SUBAPPLICATION front_fertilizer_main (* Subapplication Type *)
  (* Standard: 61499-2 *)
  (* Version 1.0, 2026-01-24, 04jul *)
  PACKAGE Main;
  IMPORT DefaultPool::Button_M1_refresh;
  IMPORT DefaultPool::Button_M1_reset;
  IMPORT DefaultPool::Button_M2_calibration_area_10a;
  IMPORT DefaultPool::Button_M2_calibration_area_1a;
  IMPORT DefaultPool::Button_M2_calibration_area_5a;
  IMPORT DefaultPool::Button_M2_start;
  IMPORT DefaultPool::Button_M4_manuel_start;
  IMPORT DefaultPool::Button_M4_manuel_stop;
  IMPORT DefaultPool::Button_W1_stop;
  IMPORT DefaultPool::Container_Picture_fertilzier_bin_empty_M1_filllevel;
  IMPORT DefaultPool::Container_Picture_fertilzier_bin_full_M1_filllevel;
  IMPORT DefaultPool::DataMask_M1;
  IMPORT DefaultPool::DataMask_M2;
  IMPORT DefaultPool::DataMask_M3;
  IMPORT DefaultPool::DataMask_M4;
  IMPORT DefaultPool::DataMask_M5;
  IMPORT DefaultPool::NumberVariable_D;
  IMPORT DefaultPool::NumberVariable_I;
  IMPORT DefaultPool::NumberVariable_P;
  IMPORT DefaultPool::NumberVariable_application_rate_percent;
  IMPORT DefaultPool::NumberVariable_engine_speed_manuel;
  IMPORT DefaultPool::NumberVariable_engine_speed_rpm;
  IMPORT DefaultPool::NumberVariable_flow_factor;
  IMPORT DefaultPool::NumberVariable_manuel_auto_speed;
  IMPORT DefaultPool::NumberVariable_selected_speed;
  IMPORT DefaultPool::NumberVariable_target_quantity;
  IMPORT DefaultPool::NumberVariable_target_quantity_calibration_run;
  IMPORT DefaultPool::OutputNumber_M1_weight;
  IMPORT DefaultPool::OutputString_M1_filllevel;
  IMPORT DefaultPool::SoftKeyMask_S1;
  IMPORT DefaultPool::SoftKeyMask_S2;
  IMPORT DefaultPool::SoftKeyMask_S3;
  IMPORT DefaultPool::SoftKeyMask_S4;
  IMPORT DefaultPool::SoftKey_100_percent;
  IMPORT DefaultPool::SoftKey_calibration_run;
  IMPORT DefaultPool::SoftKey_debug;
  IMPORT DefaultPool::SoftKey_main;
  IMPORT DefaultPool::SoftKey_minus_percent;
  IMPORT DefaultPool::SoftKey_plus_percent;
  IMPORT DefaultPool::SoftKey_settings;
  IMPORT DefaultPool::SoftKey_start;
  IMPORT DefaultPool::SoftKey_stop;
  IMPORT DefaultPool::WorkingSet_0;
  IMPORT Uebungen::const::NVS::NVS_Keys::KEY_I1_STORE;
  IMPORT Uebungen::const::NVS::NVS_Keys::KEY_I2_STORE;
  IMPORT Uebungen::const::NVS::NVS_Keys::KEY_I3_STORE;
  IMPORT Uebungen::const::NVS::NVS_Keys::SECTION_I1_STORE;
  IMPORT Uebungen::const::NVS::NVS_Keys::SECTION_I2_STORE;
  IMPORT Uebungen::const::NVS::NVS_Keys::SECTION_I3_STORE;
  IMPORT isobus::UT::Q::const::colours::COLOR_BLUE;
  IMPORT isobus::UT::Q::const::colours::COLOR_GREY;
  IMPORT isobus::UT::Q::const::colours::COLOR_RED;
  IMPORT isobus::UT::io::Button::ButtonActivationCode::BT_RELEASED_UNLATCHED;
  IMPORT isobus::UT::io::Softkey::SoftKeyActivationCode::SK_RELEASED;
  IMPORT logiBUS::io::AI::logiBUS_AI::AnalogInput_I6;
  IMPORT logiBUS::io::DI::logiBUS_DI::Input_I1;
  IMPORT logiBUS::io::DQ::logiBUS_DO::Output_Q2;
  IMPORT logiBUS::io::DQ::logiBUS_DO::Output_Q4;
  FBS
    Q_SoftKeyMask : isobus::UT::Q::Q_SoftKeyMask(u8MaskType := 1, u16DataMaskId := DataMask_M1, u16SoftKeyMaskId := SoftKeyMask_S1);
    Softkey_IE_main : isobus::UT::io::Softkey::Softkey_IE(QI := TRUE, u16ObjId := SoftKey_main, InputEvent := SK_RELEASED);
    Softkey_IE_calibration_run : isobus::UT::io::Softkey::Softkey_IE(QI := TRUE, u16ObjId := SoftKey_calibration_run, InputEvent := SK_RELEASED);
    Softkey_IE_settings : isobus::UT::io::Softkey::Softkey_IE(QI := TRUE, u16ObjId := SoftKey_settings, InputEvent := SK_RELEASED);
    Softkey_IE_debug : isobus::UT::io::Softkey::Softkey_IE(QI := TRUE, u16ObjId := SoftKey_debug, InputEvent := SK_RELEASED);
    Q_ActiveMask_DataMask_M1 : isobus::UT::Q::Q_ActiveMask(u16WorkSetId := WorkingSet_0);
    Q_NumericValue : isobus::UT::Q::Q_NumericValue(u16ObjId := NumberVariable_application_rate_percent);
    Softkey_IE_100_percent : isobus::UT::io::Softkey::Softkey_IE(QI := TRUE, u16ObjId := SoftKey_100_percent, InputEvent := SK_RELEASED);
    Softkey_IE_plus_percent : isobus::UT::io::Softkey::Softkey_IE(QI := TRUE, u16ObjId := SoftKey_plus_percent, InputEvent := SK_RELEASED);
    Softkey_IE_minus_percent : isobus::UT::io::Softkey::Softkey_IE(QI := TRUE, u16ObjId := SoftKey_minus_percent, InputEvent := SK_RELEASED);
    F_ADD : iec61131::arithmetic::F_ADD(IN2 := UDINT#278 (* Second function input *));
    F_SUB : iec61131::arithmetic::F_SUB(IN2 := UDINT#278 (* Second function input *));
    F_SEL_E_4 : eclipse4diac::utils::selection::F_SEL_E_4(IN1 := DataMask_M1, IN2 := DataMask_M2, IN3 := DataMask_M3, IN4 := DataMask_M4 (* Selectable input variable *));
    Q_ActiveMask_DataMask_M2 : isobus::UT::Q::Q_ActiveMask(u16WorkSetId := WorkingSet_0, u16NewMaskId := DataMask_M1);
    Q_SoftKeyMask_2 : isobus::UT::Q::Q_SoftKeyMask(u8MaskType := 1, u16DataMaskId := DataMask_M2, u16SoftKeyMaskId := SoftKeyMask_S2);
    Q_SoftKeyMask_3 : isobus::UT::Q::Q_SoftKeyMask(u8MaskType := 1, u16DataMaskId := DataMask_M3, u16SoftKeyMaskId := SoftKeyMask_S3);
    Q_SoftKeyMask_4 : isobus::UT::Q::Q_SoftKeyMask(u8MaskType := 1, u16DataMaskId := DataMask_M4, u16SoftKeyMaskId := SoftKeyMask_S4);
    F_SEL_E_3 : eclipse4diac::utils::selection::F_SEL_E_3(IN1 := UDINT#27780);
    NVS : eclipse4diac::storage::INI(QI := TRUE, SECTION := SECTION_I1_STORE, KEY := KEY_I1_STORE, DEFAULT_VALUE := UDINT#0);
    Q_NumericValue_1 : isobus::UT::Q::Q_NumericValue(u16ObjId := NumberVariable_application_rate_percent);
    CbVtStatus : isobus::UT::status::CbVtStatus;
    F_SEL_E_2 : eclipse4diac::utils::selection::F_SEL_E_2;
    Button_IE : isobus::UT::io::Button::Button_IE(QI := TRUE, u16ObjId := Button_M4_manuel_stop, InputEvent := BT_RELEASED_UNLATCHED);
    F_DWORD_TO_UDINT : iec61131::conversion::F_DWORD_TO_UDINT;
    InputNumber_I1 : isobus::UT::io::NumericValue::NumericValue_ID(QI := TRUE, u16ObjId := NumberVariable_flow_factor);
    INI : eclipse4diac::storage::INI(QI := TRUE, SECTION := SECTION_I2_STORE, KEY := KEY_I2_STORE, DEFAULT_VALUE := UDINT#55);
    Q_NumericValue_2 : isobus::UT::Q::Q_NumericValue(u16ObjId := NumberVariable_flow_factor);
    CbVtStatus_1 : isobus::UT::status::CbVtStatus;
    INI_1 : eclipse4diac::storage::INI(QI := TRUE, SECTION := SECTION_I3_STORE, KEY := KEY_I3_STORE, DEFAULT_VALUE := UDINT#55);
    CbVtStatus_2 : isobus::UT::status::CbVtStatus;
    F_DWORD_TO_UDINT_1 : iec61131::conversion::F_DWORD_TO_UDINT;
    InputNumber_I2 : isobus::UT::io::NumericValue::NumericValue_ID(QI := TRUE, u16ObjId := NumberVariable_target_quantity);
    Q_NumericValue_3 : isobus::UT::Q::Q_NumericValue(u16ObjId := NumberVariable_target_quantity);
    F_DINT_TO_UDINT : iec61131::conversion::F_DINT_TO_UDINT;
    F_DINT_TO_UDINT_1 : iec61131::conversion::F_DINT_TO_UDINT;
    F_DINT_TO_UDINT_2 : iec61131::conversion::F_DINT_TO_UDINT;
    logiBUS_IX : logiBUS::io::DI::logiBUS_IX(QI := True, Input := Input_I1);
    Q_StringValue : isobus::UT::Q::Q_StringValue(u16ObjId := OutputString_M1_filllevel);
    F_SEL : iec61131::selection::F_SEL(IN0 := STRING#'Tank leer', IN1 := STRING#'Tank voll');
    Q_ObjHideShow : isobus::UT::Q::Q_ObjHideShow(u16ObjId := Container_Picture_fertilzier_bin_full_M1_filllevel);
    Q_ObjHideShow_1 : isobus::UT::Q::Q_ObjHideShow(u16ObjId := Container_Picture_fertilzier_bin_empty_M1_filllevel);
    Q_BackgroundColour_3 : isobus::UT::Q::Q_BackgroundColour(u16ObjId := Button_M2_calibration_area_1a);
    Q_BackgroundColour_4 : isobus::UT::Q::Q_BackgroundColour(u16ObjId := Button_M2_calibration_area_5a);
    Q_BackgroundColour_5 : isobus::UT::Q::Q_BackgroundColour(u16ObjId := Button_M2_calibration_area_10a);
    F_SEL_E_5 : eclipse4diac::utils::selection::F_SEL_E_3(IN1 := COLOR_BLUE, IN2 := COLOR_GREY, IN3 := COLOR_GREY);
    F_SEL_E_6 : eclipse4diac::utils::selection::F_SEL_E_3(IN1 := COLOR_GREY, IN2 := COLOR_BLUE, IN3 := COLOR_GREY);
    Button_IE_1 : isobus::UT::io::Button::Button_IE(QI := TRUE, u16ObjId := Button_M2_calibration_area_1a, InputEvent := BT_RELEASED_UNLATCHED);
    Button_IE_2 : isobus::UT::io::Button::Button_IE(QI := TRUE, u16ObjId := Button_M2_calibration_area_5a, InputEvent := BT_RELEASED_UNLATCHED);
    Button_IE_3 : isobus::UT::io::Button::Button_IE(QI := TRUE, u16ObjId := Button_M2_calibration_area_10a, InputEvent := BT_RELEASED_UNLATCHED);
    F_SEL_E_7 : eclipse4diac::utils::selection::F_SEL_E_3(IN1 := COLOR_GREY, IN2 := COLOR_GREY, IN3 := COLOR_BLUE);
    Button_IE_4 : isobus::UT::io::Button::Button_IE(QI := TRUE, u16ObjId := Button_M2_start, InputEvent := BT_RELEASED_UNLATCHED);
    Q_ActiveMask_DataMask_M3 : isobus::UT::Q::Q_ActiveMask(u16WorkSetId := WorkingSet_0);
    F_SEL_E_8 : eclipse4diac::utils::selection::F_SEL_E_2(IN1 := DataMask_M5, IN2 := DataMask_M2);
    Button_IE_5 : isobus::UT::io::Button::Button_IE(QI := TRUE, u16ObjId := Button_W1_stop, InputEvent := BT_RELEASED_UNLATCHED);
    F_SEL_E_9 : eclipse4diac::utils::selection::F_SEL_E_3(IN1 := UDINT#100, IN2 := UDINT#20, IN3 := UDINT#10);
    F_DIV : iec61131::arithmetic::F_DIV;
    F_UDINT_TO_UINT : iec61131::conversion::F_UDINT_TO_UINT;
    Q_NumericValue_4 : isobus::UT::Q::Q_NumericValue(u16ObjId := NumberVariable_target_quantity_calibration_run);
    E_PERMIT : iec61499::events::E_PERMIT;
    E_SR : iec61499::events::E_SR;
    F_UDINT_TO_UINT_1 : iec61131::conversion::F_UDINT_TO_UINT;
    InputNumber_I3 : isobus::UT::io::NumericValue::NumericValue_ID(QI := TRUE, u16ObjId := NumberVariable_target_quantity);
    F_DWORD_TO_UDINT_2 : iec61131::conversion::F_DWORD_TO_UDINT;
    INI_2 : eclipse4diac::storage::INI(QI := TRUE, SECTION := SECTION_I3_STORE, KEY := KEY_I3_STORE, DEFAULT_VALUE := UDINT#55);
    Q_NumericValue_5 : isobus::UT::Q::Q_NumericValue(u16ObjId := NumberVariable_target_quantity);
    Softkey_IE_start : isobus::UT::io::Softkey::Softkey_IE(QI := TRUE, u16ObjId := SoftKey_start, InputEvent := SK_RELEASED);
    Softkey_IE_stop : isobus::UT::io::Softkey::Softkey_IE(QI := TRUE, u16ObjId := SoftKey_stop, InputEvent := SK_RELEASED);
    Q_BackgroundColour : isobus::UT::Q::Q_BackgroundColour(u16ObjId := SoftKey_start);
    Q_BackgroundColour_1 : isobus::UT::Q::Q_BackgroundColour(u16ObjId := SoftKey_stop);
    E_SR_1 : iec61499::events::E_SR;
    F_SEL_1 : iec61131::selection::F_SEL(IN0 := COLOR_BLUE, IN1 := COLOR_GREY);
    F_SEL_2 : iec61131::selection::F_SEL(IN0 := COLOR_GREY, IN1 := COLOR_RED);
    PWMOutput_Q4 : logiBUS::io::DQ::logiBUS_QD_PWM(QI := TRUE, OUT := 16#FFFFFFFF, Output := Output_Q4);
    AnalogInput_I6 : logiBUS::io::AI::logiBUS_AI_ID(QI := TRUE, Input := AnalogInput_I6, AnalogInput_hysteresis := 40);
    F_DWORD_TO_UDINT_3 : iec61131::conversion::F_DWORD_TO_UDINT;
    F_DWORD_TO_UDINT_4 : iec61131::conversion::F_DWORD_TO_UDINT;
    F_MUL : iec61131::arithmetic::F_MUL(IN2 := REAL#81.92);
    F_REAL_TO_UDINT : iec61131::conversion::F_REAL_TO_UDINT;
    F_UDINT_TO_REAL : iec61131::conversion::F_UDINT_TO_REAL;
    F_UDINT_TO_DWORD : iec61131::conversion::F_UDINT_TO_DWORD;
    F_LIMIT : iec61131::selection::F_LIMIT(MN := UDINT#0, MX := UDINT#8192);
    F_NOT : iec61131::bitwiseOperators::F_NOT;
    Button_IX : isobus::UT::io::Button::Button_IX(QI := TRUE, u16ObjId := Button_M1_reset);
    logiBUS_QX : logiBUS::io::DQ::logiBUS_QX(QI := TRUE, Output := Output_Q2);
    Q_NumericValue_6 : isobus::UT::Q::Q_NumericValue(u16ObjId := OutputNumber_M1_weight);
    E_DELAY : iec61499::events::E_DELAY(DT := T#2s);
    Button_IE_6 : isobus::UT::io::Button::Button_IE(QI := TRUE, u16ObjId := Button_M4_manuel_start, InputEvent := BT_RELEASED_UNLATCHED);
    NumericValue_ID : isobus::UT::io::NumericValue::NumericValue_ID(QI := TRUE, u16ObjId := NumberVariable_engine_speed_manuel);
    F_DWORD_TO_UDINT_5 : iec61131::conversion::F_DWORD_TO_UDINT;
    F_UDINT_TO_REAL_1 : iec61131::conversion::F_UDINT_TO_REAL;
    Q_NumericValue_7 : isobus::UT::Q::Q_NumericValue(u16ObjId := NumberVariable_engine_speed_rpm);
    F_REAL_TO_UDINT_1 : iec61131::conversion::F_REAL_TO_UDINT;
    Button_IE_7 : isobus::UT::io::Button::Button_IE(QI := TRUE, u16ObjId := Button_M1_refresh, InputEvent := BT_RELEASED_UNLATCHED);
    I_WBSD : isobus::tecu::I_WBSD(QI := TRUE);
    I_RHS : isobus::tecu::I_RHS(QI := TRUE);
    Q_NumericValue_8 : isobus::UT::Q::Q_NumericValue(u16ObjId := NumberVariable_selected_speed);
    F_UINT_TO_UDINT : iec61131::conversion::F_UINT_TO_UDINT;
    F_STRING_AS_BOOL : iec61131::conversion::F_STRING_AS_BOOL;
    F_BYTE_AS_STRING : iec61131::conversion::F_BYTE_AS_STRING;
    E_CYCLE : iec61499::events::E_CYCLE(DT := T#1s);
    NumericValue_ID_1 : isobus::UT::io::NumericValue::NumericValue_ID(QI := TRUE, u16ObjId := NumberVariable_P);
    F_DWORD_TO_UDINT_6 : iec61131::conversion::F_DWORD_TO_UDINT;
    F_UDINT_TO_REAL_2 : iec61131::conversion::F_UDINT_TO_REAL;
    NumericValue_ID_2 : isobus::UT::io::NumericValue::NumericValue_ID(QI := TRUE, u16ObjId := NumberVariable_I);
    F_DWORD_TO_UDINT_7 : iec61131::conversion::F_DWORD_TO_UDINT;
    F_UDINT_TO_REAL_3 : iec61131::conversion::F_UDINT_TO_REAL;
    NumericValue_ID_3 : isobus::UT::io::NumericValue::NumericValue_ID(QI := TRUE, u16ObjId := NumberVariable_D);
    F_DWORD_TO_UDINT_8 : iec61131::conversion::F_DWORD_TO_UDINT;
    F_UDINT_TO_REAL_4 : iec61131::conversion::F_UDINT_TO_REAL;
    NumericValue_ID_4 : isobus::UT::io::NumericValue::NumericValue_ID(QI := TRUE, u16ObjId := NumberVariable_manuel_auto_speed);
    F_DWORD_TO_UDINT_9 : iec61131::conversion::F_DWORD_TO_UDINT;
    F_UDINT_TO_REAL_5 : iec61131::conversion::F_UDINT_TO_REAL;
  END_FBS
  SUBAPPS
    Speedcontrol : Speedcontrol;
  END_SUBAPPS
  EVENT_CONNECTIONS
    Softkey_IE_minus_percent.IND TO F_SUB.REQ;
    Softkey_IE_main.IND TO F_SEL_E_4.REQ1;
    Softkey_IE_calibration_run.IND TO F_SEL_E_4.REQ2;
    Softkey_IE_settings.IND TO F_SEL_E_4.REQ3;
    Q_ActiveMask_DataMask_M2.CNF TO Q_SoftKeyMask.REQ;
    Q_SoftKeyMask.CNF TO Q_SoftKeyMask_2.REQ;
    Q_SoftKeyMask_2.CNF TO Q_SoftKeyMask_3.REQ;
    Q_SoftKeyMask_3.CNF TO Q_SoftKeyMask_4.REQ;
    Softkey_IE_plus_percent.IND TO F_ADD.REQ;
    Softkey_IE_100_percent.IND TO F_SEL_E_3.REQ1;
    NVS.GETO TO Q_NumericValue_1.REQ;
    CbVtStatus.IND TO Q_NumericValue_1.REQ;
    NVS.INITO TO NVS.GET;
    F_SEL_E_2.CNF TO Q_NumericValue.REQ;
    Q_NumericValue_1.CNF TO F_SEL_E_2.REQ2;
    InputNumber_I1.IND TO F_DWORD_TO_UDINT.REQ;
    F_DWORD_TO_UDINT.CNF TO INI.SET;
    INI.GETO TO Q_NumericValue_2.REQ;
    CbVtStatus_1.IND TO Q_NumericValue_2.REQ;
    INI.INITO TO INI.GET;
    CbVtStatus_2.IND TO Q_NumericValue_3.REQ;
    INI_1.INITO TO INI_1.GET;
    F_DWORD_TO_UDINT_1.CNF TO INI_1.SET;
    INI_1.GETO TO Q_NumericValue_3.REQ;
    InputNumber_I2.IND TO F_DWORD_TO_UDINT_1.REQ;
    F_SUB.CNF TO F_DINT_TO_UDINT.REQ;
    F_DINT_TO_UDINT.CNF TO F_SEL_E_3.REQ3;
    F_DINT_TO_UDINT_1.CNF TO F_SEL_E_3.REQ2;
    F_ADD.CNF TO F_DINT_TO_UDINT_1.REQ;
    F_SEL_E_3.CNF TO F_DINT_TO_UDINT_2.REQ;
    F_DINT_TO_UDINT_2.CNF TO F_SEL_E_2.REQ1;
    F_DINT_TO_UDINT_2.CNF TO NVS.SET;
    logiBUS_IX.IND TO F_SEL.REQ;
    F_SEL.CNF TO Q_StringValue.REQ;
    logiBUS_IX.IND TO Q_ObjHideShow.REQ;
    Button_IE_1.IND TO F_SEL_E_5.REQ1;
    Button_IE_1.IND TO F_SEL_E_6.REQ1;
    Button_IE_2.IND TO F_SEL_E_5.REQ2;
    Button_IE_2.IND TO F_SEL_E_6.REQ2;
    Button_IE_3.IND TO F_SEL_E_5.REQ3;
    Button_IE_3.IND TO F_SEL_E_6.REQ3;
    Button_IE_3.IND TO F_SEL_E_7.REQ3;
    Button_IE_2.IND TO F_SEL_E_7.REQ2;
    Button_IE_1.IND TO F_SEL_E_7.REQ1;
    F_SEL_E_5.CNF TO Q_BackgroundColour_3.REQ;
    F_SEL_E_6.CNF TO Q_BackgroundColour_4.REQ;
    Q_ObjHideShow_1.CNF TO Q_ObjHideShow.REQ;
    F_SEL_E_7.CNF TO Q_BackgroundColour_5.REQ;
    F_SEL_E_4.CNF TO Q_ActiveMask_DataMask_M1.REQ;
    Button_IE_5.IND TO F_SEL_E_8.REQ2;
    Softkey_IE_debug.IND TO F_SEL_E_4.REQ4;
    F_SEL_E_8.CNF TO Q_ActiveMask_DataMask_M3.REQ;
    Button_IE_1.IND TO F_SEL_E_9.REQ1;
    Button_IE_2.IND TO F_SEL_E_9.REQ2;
    Button_IE_3.IND TO F_SEL_E_9.REQ3;
    F_SEL_E_9.CNF TO F_UDINT_TO_UINT.REQ;
    F_DIV.CNF TO Q_NumericValue_4.REQ;
    Button_IE_4.IND TO E_PERMIT.EI;
    E_PERMIT.EO TO F_SEL_E_8.REQ1;
    F_SEL_E_9.CNF TO E_SR.S;
    F_UDINT_TO_UINT.CNF TO INI_1.GET;
    INI_1.GETO TO F_UDINT_TO_UINT_1.REQ;
    F_UDINT_TO_UINT_1.CNF TO F_DIV.REQ;
    INI_2.GETO TO Q_NumericValue_5.REQ;
    InputNumber_I3.IND TO F_DWORD_TO_UDINT_2.REQ;
    F_DWORD_TO_UDINT_2.CNF TO INI_2.SET;
    INI_2.INITO TO INI_2.GET;
    Softkey_IE_start.IND TO E_SR_1.S;
    Softkey_IE_stop.IND TO E_SR_1.R;
    E_SR_1.EO TO F_SEL_1.REQ;
    E_SR_1.EO TO F_SEL_2.REQ;
    F_SEL_2.CNF TO Q_BackgroundColour_1.REQ;
    F_SEL_1.CNF TO Q_BackgroundColour.REQ;
    Q_ActiveMask_DataMask_M1.CNF TO E_SR_1.R;
    AnalogInput_I6.IND TO F_DWORD_TO_UDINT_3.REQ;
    InputNumber_I1.IND TO F_DWORD_TO_UDINT_4.REQ;
    InputNumber_I1.INITO TO F_DWORD_TO_UDINT_4.REQ;
    F_MUL.CNF TO F_REAL_TO_UDINT.REQ;
    F_DWORD_TO_UDINT_4.CNF TO F_UDINT_TO_REAL.REQ;
    F_UDINT_TO_REAL.CNF TO F_MUL.REQ;
    F_UDINT_TO_DWORD.CNF TO PWMOutput_Q4.REQ;
    F_REAL_TO_UDINT.CNF TO F_LIMIT.REQ;
    F_LIMIT.CNF TO F_UDINT_TO_DWORD.REQ;
    F_NOT.CNF TO Q_ObjHideShow_1.REQ;
    logiBUS_IX.IND TO F_NOT.REQ;
    Button_IX.IND TO logiBUS_QX.REQ;
    F_DWORD_TO_UDINT_3.CNF TO Q_NumericValue_6.REQ;
    Q_ActiveMask_DataMask_M2.INITO TO E_DELAY.START;
    E_DELAY.EO TO Q_ActiveMask_DataMask_M2.REQ;
    E_DELAY.EO TO logiBUS_IX.REQ;
    Softkey_IE_start.IND TO Speedcontrol.START;
    Softkey_IE_stop.IND TO Speedcontrol.STOP;
    Button_IE.IND TO Speedcontrol.M_STOP;
    Button_IE_6.IND TO Speedcontrol.M_START;
    NumericValue_ID.IND TO F_DWORD_TO_UDINT_5.REQ;
    F_DWORD_TO_UDINT_5.CNF TO F_UDINT_TO_REAL_1.REQ;
    F_UDINT_TO_REAL_1.CNF TO Speedcontrol.REQ_PID;
    Speedcontrol.CNF_SPEED TO F_REAL_TO_UDINT_1.REQ;
    F_REAL_TO_UDINT_1.CNF TO Q_NumericValue_7.REQ;
    Button_IE_7.IND TO Q_ActiveMask_DataMask_M2.REQ;
    F_UINT_TO_UDINT.CNF TO Q_NumericValue_8.REQ;
    I_WBSD.IND TO F_UINT_TO_UDINT.REQ;
    F_BYTE_AS_STRING.CNF TO F_STRING_AS_BOOL.REQ;
    I_WBSD.INITO TO E_CYCLE.START;
    E_CYCLE.EO TO I_RHS.INIT;
    I_RHS.INITO TO F_BYTE_AS_STRING.REQ;
    NumericValue_ID_1.IND TO F_DWORD_TO_UDINT_6.REQ;
    F_DWORD_TO_UDINT_6.CNF TO F_UDINT_TO_REAL_2.REQ;
    F_UDINT_TO_REAL_2.CNF TO Speedcontrol.REQ_PID;
    NumericValue_ID_2.IND TO F_DWORD_TO_UDINT_7.REQ;
    F_UDINT_TO_REAL_3.CNF TO Speedcontrol.REQ_PID;
    F_DWORD_TO_UDINT_7.CNF TO F_UDINT_TO_REAL_3.REQ;
    NumericValue_ID_3.IND TO F_DWORD_TO_UDINT_8.REQ;
    F_UDINT_TO_REAL_4.CNF TO Speedcontrol.REQ_PID;
    F_DWORD_TO_UDINT_8.CNF TO F_UDINT_TO_REAL_4.REQ;
    NumericValue_ID_4.IND TO F_DWORD_TO_UDINT_9.REQ;
    F_UDINT_TO_REAL_5.CNF TO Speedcontrol.REQ_PID;
    F_DWORD_TO_UDINT_9.CNF TO F_UDINT_TO_REAL_5.REQ;
  END_CONNECTIONS
  DATA_CONNECTIONS
    Q_NumericValue.u32OldValue TO F_ADD.IN1;
    Q_NumericValue.u32OldValue TO F_SUB.IN1;
    NVS.VALUEO TO Q_NumericValue_1.u32NewValue;
    F_SEL_E_2.OUT TO Q_NumericValue.u32NewValue;
    Q_NumericValue_1.u32OldValue TO F_SEL_E_2.IN2;
    InputNumber_I1.IN TO F_DWORD_TO_UDINT.IN;
    F_DWORD_TO_UDINT.OUT TO INI.VALUE;
    INI.VALUEO TO Q_NumericValue_2.u32NewValue;
    F_DWORD_TO_UDINT_1.OUT TO INI_1.VALUE;
    INI_1.VALUEO TO Q_NumericValue_3.u32NewValue;
    InputNumber_I2.IN TO F_DWORD_TO_UDINT_1.IN;
    F_SUB.OUT TO F_DINT_TO_UDINT.IN;
    F_DINT_TO_UDINT.OUT TO F_SEL_E_3.IN3;
    F_DINT_TO_UDINT_1.OUT TO F_SEL_E_3.IN2;
    F_ADD.OUT TO F_DINT_TO_UDINT_1.IN;
    F_SEL_E_3.OUT TO F_DINT_TO_UDINT_2.IN;
    F_DINT_TO_UDINT_2.OUT TO F_SEL_E_2.IN1;
    F_DINT_TO_UDINT_2.OUT TO NVS.VALUE;
    F_SEL.OUT TO Q_StringValue.pau8String;
    logiBUS_IX.IN TO F_SEL.G;
    logiBUS_IX.IN TO Q_ObjHideShow.qVisible;
    F_SEL_E_5.OUT TO Q_BackgroundColour_3.u8Colour;
    F_SEL_E_6.OUT TO Q_BackgroundColour_4.u8Colour;
    F_SEL_E_7.OUT TO Q_BackgroundColour_5.u8Colour;
    F_SEL_E_4.OUT TO Q_ActiveMask_DataMask_M1.u16NewMaskId;
    F_SEL_E_8.OUT TO Q_ActiveMask_DataMask_M3.u16NewMaskId;
    F_SEL_E_9.OUT TO F_UDINT_TO_UINT.IN;
    F_UDINT_TO_UINT.OUT TO F_DIV.IN2;
    F_DIV.OUT TO Q_NumericValue_4.u32NewValue;
    E_SR.Q TO E_PERMIT.PERMIT;
    INI_1.VALUEO TO F_UDINT_TO_UINT_1.IN;
    F_UDINT_TO_UINT_1.OUT TO F_DIV.IN1;
    INI_2.VALUEO TO Q_NumericValue_5.u32NewValue;
    InputNumber_I3.IN TO F_DWORD_TO_UDINT_2.IN;
    F_DWORD_TO_UDINT_2.OUT TO INI_2.VALUE;
    E_SR_1.Q TO F_SEL_1.G;
    E_SR_1.Q TO F_SEL_2.G;
    F_SEL_1.OUT TO Q_BackgroundColour.u8Colour;
    F_SEL_2.OUT TO Q_BackgroundColour_1.u8Colour;
    AnalogInput_I6.IN TO F_DWORD_TO_UDINT_3.IN;
    InputNumber_I1.IN TO F_DWORD_TO_UDINT_4.IN;
    F_MUL.OUT TO F_REAL_TO_UDINT.IN;
    F_DWORD_TO_UDINT_4.OUT TO F_UDINT_TO_REAL.IN;
    F_UDINT_TO_REAL.OUT TO F_MUL.IN1;
    F_UDINT_TO_DWORD.OUT TO PWMOutput_Q4.OUT;
    F_REAL_TO_UDINT.OUT TO F_LIMIT.IN;
    F_LIMIT.OUT TO F_UDINT_TO_DWORD.IN;
    logiBUS_IX.IN TO F_NOT.IN;
    F_NOT.OUT TO Q_ObjHideShow_1.qVisible;
    Button_IX.IN TO logiBUS_QX.OUT;
    F_DWORD_TO_UDINT_3.OUT TO Q_NumericValue_6.u32NewValue;
    NumericValue_ID.IN TO F_DWORD_TO_UDINT_5.IN;
    F_UDINT_TO_REAL_1.OUT TO Speedcontrol.M_INPUT;
    F_DWORD_TO_UDINT_5.OUT TO F_UDINT_TO_REAL_1.IN;
    Speedcontrol.OUTPUT_SPEED TO F_REAL_TO_UDINT_1.IN;
    F_REAL_TO_UDINT_1.OUT TO Q_NumericValue_7.u32NewValue;
    F_UINT_TO_UDINT.OUT TO Q_NumericValue_8.u32NewValue;
    I_WBSD.WHEELBASEDMACHINESPEED TO F_UINT_TO_UDINT.IN;
    I_RHS.REAR_HITCH_WORK_INDICATION TO F_BYTE_AS_STRING.IN;
    F_BYTE_AS_STRING.OUT TO F_STRING_AS_BOOL.IN;
    NumericValue_ID_1.IN TO F_DWORD_TO_UDINT_6.IN;
    F_DWORD_TO_UDINT_6.OUT TO F_UDINT_TO_REAL_2.IN;
    F_DWORD_TO_UDINT_7.OUT TO F_UDINT_TO_REAL_3.IN;
    NumericValue_ID_2.IN TO F_DWORD_TO_UDINT_7.IN;
    F_DWORD_TO_UDINT_8.OUT TO F_UDINT_TO_REAL_4.IN;
    NumericValue_ID_3.IN TO F_DWORD_TO_UDINT_8.IN;
    F_DWORD_TO_UDINT_9.OUT TO F_UDINT_TO_REAL_5.IN;
    NumericValue_ID_4.IN TO F_DWORD_TO_UDINT_9.IN;
    F_UDINT_TO_REAL_2.OUT TO Speedcontrol.P;
    F_UDINT_TO_REAL_3.OUT TO Speedcontrol.I;
    F_UDINT_TO_REAL_4.OUT TO Speedcontrol.DIF;
    F_UDINT_TO_REAL_5.OUT TO Speedcontrol.SET_SPEED;
  END_CONNECTIONS
END_SUBAPPLICATION
